# EPICS autosave request: ADQImaging/App/Db/qimaging_settings.req
file "ADBase_settings.req", P=$(P), R=$(R)
$(P)$(R)qReadoutSpeed
$(P)$(R)qOffset
$(P)$(R)qImageFormat
$(P)$(R)qCoolerActive
